(* IEC 61131-3 sources: Automatisierte-Tank-und-Pumpensteuerung/sps/function_blocks, 7 files *)

(* ---- FB_Alarm.st ---- *)
(*
    sps/function_blocks/FB_Alarm.st
    Generischer Alarm-Baustein.

    Jede Alarminstanz erhaelt eine feste Kennung und Prioritaet sowie die
    ausloesende Bedingung. Der Alarm wird gespeichert (latch) und kann mit
    einem Sammelreset (Flanke) quittiert/zurueckgesetzt werden.
*)

FUNCTION_BLOCK FB_Alarm
VAR_INPUT
    xTrigger : BOOL;        (* Ausloesende Bedingung *)
    xReset   : BOOL;        (* Sammelreset (Flanke vom PLC_PRG) *)
    id       : E_AlarmId;
    severity : E_Severity;
    xDelay   : BOOL;        (* optionale Verzoegerung aktiv *)
    tDelayMs : DINT;        (* Verzoegerungszeit *)
END_VAR
VAR_OUTPUT
    xActive      : BOOL;    (* Bedingung liegt aktuell an *)
    xLatched     : BOOL;    (* gespeichert, bis Reset *)
    xAcknowledged: BOOL;    (* quittiert *)
END_VAR
VAR
    fbDelay : FB_TON;
    xCond   : BOOL;
END_VAR
    (* optionale Einschaltverzoegerung *)
    IF xDelay THEN
        fbDelay(IN := xTrigger, PT := tDelayMs);
        xCond := fbDelay.Q;
    ELSE
        fbDelay(IN := FALSE, PT := tDelayMs);
        xCond := xTrigger;
    END_IF

    (* Speichern (latch) *)
    IF xCond THEN
        xLatched := TRUE;
    END_IF

    xActive := xCond;

    (* Reset: nur wenn Bedingung nicht mehr anliegt, wird der Alarm geloescht *)
    IF xReset THEN
        xAcknowledged := TRUE;
        IF NOT xCond THEN
            xLatched := FALSE;
            xAcknowledged := FALSE;
        END_IF
    END_IF
END_FUNCTION_BLOCK

(* ---- FB_ModeManager.st ---- *)
(*
    sps/function_blocks/FB_ModeManager.st
    Betriebsarten- und Tasterauswertung.

    Aufgaben:
      - Betriebsart aus Wahlschalter (AUTO / HAND)
      - Start/Stop als gespeicherter Laufwunsch (Flankenauswertung)
      - Reset-Sammelimpuls (Flanke)
*)

FUNCTION_BLOCK FB_ModeManager
VAR_INPUT
    xModeAuto : BOOL;       (* Wahlschalter *)
    xStartBtn : BOOL;
    xStopBtn  : BOOL;
    xResetBtn : BOOL;
END_VAR
VAR_OUTPUT
    eMode       : E_Mode;
    xRunRequest : BOOL;     (* Laufwunsch, gespeichert *)
    xStartPulse : BOOL;     (* Flanke Start *)
    xStopPulse  : BOOL;     (* Flanke Stop *)
    xResetPulse : BOOL;     (* Flanke Reset *)
END_VAR
VAR
    fbStart : FB_R_TRIG;
    fbStop  : FB_R_TRIG;
    fbReset : FB_R_TRIG;
END_VAR
    fbStart(CLK := xStartBtn);
    fbStop(CLK := xStopBtn);
    fbReset(CLK := xResetBtn);

    xStartPulse := fbStart.Q;
    xStopPulse  := fbStop.Q;
    xResetPulse := fbReset.Q;

    IF xModeAuto THEN
        eMode := E_Mode#MODE_AUTO;
    ELSE
        eMode := E_Mode#MODE_MANUAL;
    END_IF

    (* Laufwunsch speichern *)
    IF xStartPulse THEN
        xRunRequest := TRUE;
    END_IF
    IF xStopPulse THEN
        xRunRequest := FALSE;
    END_IF
END_FUNCTION_BLOCK

(* ---- FB_Pump.st ---- *)
(*
    sps/function_blocks/FB_Pump.st
    Pumpensteuerung mit Sicherheitsfreigabe und Rueckmeldungsueberwachung.

    Verriegelungen:
      - Ausgang nur bei xEnable (Freigabe aus FB_Safety) und xCommand
      - bei Ueberlast (xOverload) -> Störung, Ausgang AUS
      - fehlende Lauf-Rueckmeldung nach Ablauf von tFeedbackMs -> Stoerung
    Stoerungen werden gespeichert und durch xReset (Flanke) zurueckgesetzt.
*)

FUNCTION_BLOCK FB_Pump
VAR_INPUT
    xCommand    : BOOL;     (* Betrieb angefordert *)
    xEnable     : BOOL;     (* Freigabe (Verriegelung) *)
    xFeedback   : BOOL;     (* Rueckmeldung "Pumpe laeuft" *)
    xOverload   : BOOL;     (* Motorschutz/Fault vom Feld *)
    xReset      : BOOL;     (* Stoerungsreset (Flanke) *)
    tFeedbackMs : DINT;     (* Ueberwachungszeit *)
END_VAR
VAR_OUTPUT
    xRun           : BOOL;  (* Pumpenausgang *)
    xFault         : BOOL;  (* gespeicherte Stoerung *)
    xFeedbackFault : BOOL;  (* Rueckmeldung ausgeblieben *)
    xFeedbackOK    : BOOL;  (* Rueckmeldung plausibel *)
END_VAR
VAR
    fbFeedback : FB_TON;
END_VAR
    (* Reset der gespeicherten Stoerung *)
    IF xReset THEN
        xFault := FALSE;
        xFeedbackFault := FALSE;
    END_IF

    (* Ueberlast ist eine sofortige, speichernde Stoerung *)
    IF xOverload THEN
        xFault := TRUE;
    END_IF

    (* Ausgang nur bei Anforderung + Freigabe + keiner Stoerung *)
    xRun := xCommand AND xEnable AND NOT xFault;

    (* Ueberwachung der Lauf-Rueckmeldung *)
    fbFeedback(IN := xRun AND NOT xFeedback, PT := tFeedbackMs);
    xFeedbackOK := xRun AND xFeedback;
    IF xRun AND NOT xFeedback AND fbFeedback.Q THEN
        xFeedbackFault := TRUE;
        xFault := TRUE;
        xRun := FALSE;
    END_IF
END_FUNCTION_BLOCK

(* ---- FB_Safety.st ---- *)
(*
    sps/function_blocks/FB_Safety.st
    Sicherheits- und Verriegelungslogik.

    Zentrale Freigaben fuer Pumpe, Zulauf und Ablauf. In einer realen Anlage
    schaltet ein Sicherheitsschaltgeraet (z. B. PNOZ) den Not-Aus allpolig ab;
    hier ist diese Abschaltung logisch nachgebildet.

    Die Aktor-Bausteine (FB_Pump, FB_Valve) setzen diese Freigaben zusaetzlich
    zu ihren eigenen Verriegelungen durch.
*)

FUNCTION_BLOCK FB_Safety
VAR_INPUT
    xEStop              : BOOL; (* Not-Aus aktiv *)
    xPumpOverload       : BOOL; (* Motorueberlast *)
    xPumpFeedbackFault  : BOOL; (* Pumpen-Rueckmeldung fehlt *)
    xValveFault         : BOOL; (* Ventilstellungsfehler *)
    xSensorError        : BOOL; (* unplausible Sensorik *)
    xCriticalHigh       : BOOL; (* kritisch hoher Füllstand *)
    xCriticalLow        : BOOL; (* kritisch niedriger Füllstand *)
END_VAR
VAR_OUTPUT
    xSafe        : BOOL;        (* Grundfreigabe (kein Not-Aus) *)
    xPumpEnable  : BOOL;        (* Freigabe Pumpe *)
    xFillEnable  : BOOL;        (* Freigabe Zulaufventil *)
    xDrainEnable : BOOL;        (* Freigabe Ablaufventil *)
    xAnyFault    : BOOL;        (* Sammelstoerung *)
END_VAR
    (* Not-Aus hebt jede Freigabe auf *)
    xSafe := NOT xEStop;

    (* Sammelstoerung (fuehrt in den FAULT-Zustand) *)
    xAnyFault := xPumpOverload OR xPumpFeedbackFault OR xValveFault
                 OR xSensorError OR xCriticalHigh;

    (* Pumpe: keine Freigabe bei Ueberlast/Rueckmeldungsfehler/kritisch niedrig *)
    xPumpEnable  := xSafe AND NOT xPumpOverload AND NOT xPumpFeedbackFault
                    AND NOT xCriticalLow AND NOT xSensorError;

    (* Zulauf: keine Freigabe bei kritisch hoch / Ventilfehler / Sensorfehler *)
    xFillEnable  := xSafe AND NOT xCriticalHigh AND NOT xValveFault
                    AND NOT xSensorError;

    (* Ablauf: nur Grundfreigabe und plausible Sensorik *)
    xDrainEnable := xSafe AND NOT xSensorError;
END_FUNCTION_BLOCK

(* ---- FB_Stats.st ---- *)
(*
    sps/function_blocks/FB_Stats.st
    Betriebsstatistik: Zyklen, Betriebszeit, Pumpenlaufzeit, Fuellzyklen.
*)

FUNCTION_BLOCK FB_Stats
VAR_INPUT
    xProcessRunning : BOOL;  (* Prozess aktiv (FILLING/PUMPING) *)
    xPumpRunning    : BOOL;  (* Pumpenausgang *)
    xFillDone       : BOOL;  (* Flanke: Fuellzyklus abgeschlossen *)
END_VAR
VAR_OUTPUT
    diCycles        : DINT;  (* Zyklen gesamt *)
    diRunTimeMs     : DINT;  (* Betriebszeit Prozess (ms) *)
    diPumpRunTimeMs : DINT;  (* Pumpenlaufzeit (ms) *)
    diFillCycles    : DINT;  (* abgeschlossene Fuellzyklen *)
END_VAR
VAR
    fbFillDone : FB_R_TRIG;
END_VAR
    diCycles := diCycles + 1;

    IF xProcessRunning THEN
        diRunTimeMs := diRunTimeMs + SCAN_PERIOD_MS;
    END_IF
    IF xPumpRunning THEN
        diPumpRunTimeMs := diPumpRunTimeMs + SCAN_PERIOD_MS;
    END_IF

    fbFillDone(CLK := xFillDone);
    IF fbFillDone.Q THEN
        diFillCycles := diFillCycles + 1;
    END_IF
END_FUNCTION_BLOCK

(* ---- FB_TankControl.st ---- *)
(*
    sps/function_blocks/FB_TankControl.st
    Füllstandsauswertung.

    Aufgaben:
      - Skalierung des analogen Rohwerts (0..27648) in Prozent (0..100)
      - Plausibilitaetspruefung (Grenzwert-Widerspruch, Bereichsfehler)
      - Ableitung der Grenzwertmeldungen (High, Critical, Critical-Low)
      - Fuellbedarf mit Hysterese (Start 30 %, Stopp 80 %)
*)

FUNCTION_BLOCK FB_TankControl
VAR_INPUT
    iwRaw         : INT;    (* analoger Rohwert *)
    xLowLevel     : BOOL;   (* digitaler Grenzwertschalter Low *)
    xHighLevel    : BOOL;   (* digitaler Grenzwertschalter High *)
    xVeryHighLevel: BOOL;   (* digitaler Grenzwertschalter Very-High *)
END_VAR
VAR_OUTPUT
    rLevelPct     : REAL;   (* Füllstand in % *)
    xRawOutOfRange: BOOL;   (* Rohwert ausserhalb 0..27648 *)
    xSensorError  : BOOL;   (* unplausible Sensorinformation *)
    xHighAlarm    : BOOL;   (* >= 90 % *)
    xCriticalHigh : BOOL;   (* >= 95 % *)
    xCriticalLow  : BOOL;   (* <= 10 % *)
    xFillDemand   : BOOL;   (* Fuellen erforderlich (mit Hysterese) *)
    xLowSensor    : BOOL;   (* digitaler Low-Grenzwert *)
END_VAR
VAR
    rLastValid  : REAL;     (* letzter gueltiger Messwert *)
    initialized : BOOL;
END_VAR
    (* --- Plausibilitaet des Rohwerts --- *)
    xRawOutOfRange := (iwRaw < RAW_MIN) OR (iwRaw > RAW_MAX);
    (* Widerspruch: Low- und High-Grenzwert gleichzeitig aktiv *)
    xSensorError := (xLowLevel AND xHighLevel) OR xRawOutOfRange;

    (* --- Skalierung Rohwert -> Engineering Unit [%] --- *)
    IF xRawOutOfRange THEN
        (* ungueltiger Wert: letzten gueltigen Messwert halten *)
        rLevelPct := rLastValid;
    ELSE
        rLevelPct := EU_MIN +
                     (INT_TO_REAL(iwRaw - RAW_MIN) / INT_TO_REAL(RAW_MAX - RAW_MIN)) *
                     (EU_MAX - EU_MIN);
        rLevelPct := LIMIT_REAL(rLevelPct, EU_MIN, EU_MAX);
        rLastValid := rLevelPct;
    END_IF

    (* --- Grenzwerte (analog ODER digital) --- *)
    xLowSensor    := xLowLevel;
    xHighAlarm    := (rLevelPct >= LVL_HIGH_ALARM_PCT) OR xHighLevel;
    xCriticalHigh := (rLevelPct >= LVL_CRITICAL_PCT) OR xVeryHighLevel;
    xCriticalLow  := rLevelPct <= LVL_CRITICAL_LOW_PCT;

    (* --- Fuellbedarf mit Hysterese (Start 30 %, Stopp 80 %) --- *)
    IF NOT initialized THEN
        xFillDemand := rLevelPct < LVL_FILL_START_PCT;
        initialized := TRUE;
    END_IF
    IF rLevelPct <= LVL_FILL_START_PCT THEN
        xFillDemand := TRUE;
    ELSIF rLevelPct >= LVL_FILL_STOP_PCT THEN
        xFillDemand := FALSE;
    END_IF
END_FUNCTION_BLOCK

(* ---- FB_Valve.st ---- *)
(*
    sps/function_blocks/FB_Valve.st
    Ventilsteuerung mit Endlagen-Rueckmeldung.

    Verriegelungen:
      - Ausgang nur bei xEnable (Freigabe) und xCommand
      - bleibt die Offen-Rueckmeldung nach tFeedbackMs aus, obwohl das Ventil
        geoeffnet werden soll, wird eine Störung erzeugt (Stellungsfehler)
    Stoerungen werden gespeichert und durch xReset (Flanke) zurueckgesetzt.
*)

FUNCTION_BLOCK FB_Valve
VAR_INPUT
    xCommand        : BOOL;  (* Offen angefordert *)
    xEnable         : BOOL;  (* Freigabe (Verriegelung) *)
    xFeedbackOpen   : BOOL;  (* Rueckmeldung "offen" *)
    xFeedbackClosed : BOOL;  (* Rueckmeldung "geschlossen" *)
    xReset          : BOOL;  (* Stoerungsreset (Flanke) *)
    tFeedbackMs     : DINT;  (* Ueberwachungszeit *)
END_VAR
VAR_OUTPUT
    xOpen          : BOOL;   (* Ventilausgang *)
    xFault         : BOOL;   (* gespeicherte Stellungsstoerung *)
    xFeedbackOK    : BOOL;   (* Endlage passt zum Befehl *)
END_VAR
VAR
    fbFeedback : FB_TON;
END_VAR
    IF xReset THEN
        xFault := FALSE;
    END_IF

    xOpen := xCommand AND xEnable AND NOT xFault;

    (* Rueckmeldung pruefen: offen gefordert, aber nicht "offen" gemeldet *)
    fbFeedback(IN := xOpen AND NOT xFeedbackOpen, PT := tFeedbackMs);
    xFeedbackOK := (xOpen AND xFeedbackOpen) OR ((NOT xOpen) AND xFeedbackClosed);
    IF xOpen AND NOT xFeedbackOpen AND fbFeedback.Q THEN
        xFault := TRUE;
        xOpen := FALSE;
    END_IF
END_FUNCTION_BLOCK
